FUNCTION_BLOCK AX_BLINK_TRAIN (* Simulates a blinking signal (turning on and off for specific durations), with a limited N *)
  (* Standard: 61499-1; Description: Copyright (c) 2025 HR Agrartechnik GmbH This program and the accompanying materials are made available under the terms of the Eclipse Public License 2.0 which is available at https://www.eclipse.org/legal/epl-2.0/ SPDX-License-Identifier: EPL-2.0 was a little inspired by this FUNCTION_BLOCK BLINK: https://content.helpme-codesys.com/en/libs/Util/Current/Signals/BLINK.html BUT while CODESYS keeps the last State, this FB return to FALSE on STOP. *)
  (* Version 3.0, 2025-04-14, Patrick Aigner, changed package *)
  (* Version 1.0, 2025-02-15, Franz Höpfinger, HR Agrartechnik GmbH, initial API and implementation and/or initial documentation *)
  PACKAGE adapter::events::unidirectional::signals;
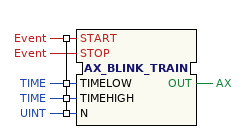
  EVENT_INPUT
    START WITH TIMELOW, TIMEHIGH, N; (* Start the perodic generation of events *)
    STOP; (* Stop the generation of events *)
  END_EVENT
  VAR_INPUT
    TIMELOW : TIME; (* Time for OUT to be FALSE *)
    TIMEHIGH : TIME; (* Time for OUT to be TRUE *)
    N : UINT; (* Number of events to generate *)
  END_VAR
  PLUGS
    OUT : adapter::types::unidirectional::AX; (* Output value, starts with FALSE and switches between TRUE and FALSE for the given high and low times *)
  END_PLUGS
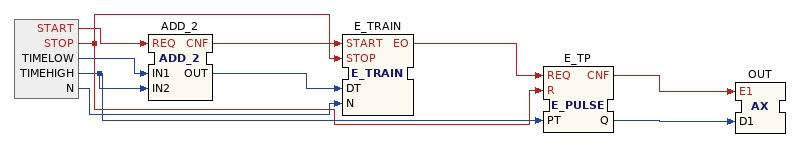
  FBS
    E_TP : iec61499::events::timers::E_PULSE;
    E_TRAIN : iec61499::events::E_TRAIN;
    ADD_2 : iec61131::arithmetic::ADD_2;
  END_FBS
  EVENT_CONNECTIONS
    E_TRAIN.EO TO E_TP.REQ;
    START TO ADD_2.REQ;
    ADD_2.CNF TO E_TRAIN.START;
    STOP TO E_TRAIN.STOP;
    STOP TO E_TP.R;
    E_TP.CNF TO OUT.E1;
  END_CONNECTIONS
  DATA_CONNECTIONS
    ADD_2.OUT TO E_TRAIN.DT;
    TIMELOW TO ADD_2.IN1;
    TIMEHIGH TO ADD_2.IN2;
    TIMEHIGH TO E_TP.PT;
    N TO E_TRAIN.N;
    E_TP.Q TO OUT.D1;
  END_CONNECTIONS
END_FUNCTION_BLOCK
